FUNCTION TryConvert_TOD_TO_DINT : BOOL
VAR_INPUT
	in : TOD;
	out : REFERENCE TO DINT;
END_VAR

out := TOD_TO_DINT(in);
TryConvert_TOD_TO_DINT := TRUE;

END_FUNCTION

(* stored: Version 1.1.0.1, ProductVersion 3.1.4024.12
   POU TryConvert_TOD_TO_DINT: Id {f727dace-17cc-4a9f-b610-ec8d15b29fc3}, SpecialFunc None *)
